PROGRAM conveyor1
VAR
	bStatus: BOOL;
	bSensor2: BOOL;
	bSensor1: BOOL;
	bAlimentador1: BOOL;
	intCaseConveyor : INT;
	bButtonReset: BOOL;
	timer1, timer2, timer3,timer4 : TON;
	bConvFowar1: BOOL;
	bMachineCenterOpen: BOOL;
	bMachineCenterBusy: BOOL;
	bStartMachineCenter: BOOL;
	wMachineProgress: WORD;
END_VAR

bStatus := tags.bAutoMan.Q1;
bSensor1 := GVL.mb_Output_Coils[10];
bSensor2 := GVL.mb_Output_Coils[11];
bButtonReset := gvl.mb_Output_Coils[2];
bMachineCenterOpen := gvl.mb_Output_Coils[12];
bMachineCenterBusy := gvl.mb_Output_Coils[13];
wMachineProgress := gvl.mb_Output_Registers[0];


GVL.mb_Input_Coils[10] := bAlimentador1;
GVL.mb_Input_Coils[11] := bConvFowar1;
GVL.mb_Input_Coils[12] := bStartMachineCenter;

timer1(PT:= T#1S);
timer2(PT:= T#1S);
timer3(PT:= T#1S);


IF NOT bStatus THEN
	intCaseConveyor := 0;
END_IF

IF intCaseConveyor = 40 THEN
	timer2(IN := TRUE);
ELSE
	timer2(IN := FALSE);
END_IF

IF intCaseConveyor = 50 THEN
	timer3(IN := TRUE);
ELSE
	timer3(IN := FALSE);
END_IF

CASE intCaseConveyor OF
	00: timer1(IN:= FALSE);
		timer4(IN:= FALSE);
		bConvFowar1 := FALSE;
		bStartMachineCenter := False;
		IF bStatus THEN
			IF bSensor1 THEN
				intCaseConveyor := 10;
			ELSE
				intCaseConveyor := 20;
			END_IF
		END_IF
	10: IF bSensor1 THEN
			bAlimentador1 := TRUE;
		ELSE
			bAlimentador1 := FALSE;
			intCaseConveyor := 20;
		END_IF
	20: timer1(in:= TRUE);
		IF timer1.Q THEN
			bConvFowar1 := TRUE;
			intCaseConveyor := 30;
		END_IF;
	30: IF NOT bsensor2 THEN
			bConvFowar1 := FALSE;
				intCaseConveyor := 40;
		END_IF
		
	40: IF timer2.Q AND NOT bMachineCenterbusy  THEN
			bConvFowar1 := TRUE;
			IF bSensor2 THEN
				intCaseConveyor := 50;
			END_IF
		END_IF
	50: IF timer3.Q THEN
			bStartMachineCenter := TRUE;
			timer4(IN:= TRUE, PT:= T#300MS);
			IF timer4.Q THEN
				intCaseConveyor := 0;
			END_IF
		END_IF
		
END_CASE

END_PROGRAM

(* stored: Version 1.1.0.1, ProductVersion 3.1.4024.12
   POU conveyor1: Id {a9931d23-820b-42ce-abd7-93b93010757f}, SpecialFunc None *)
